{attribute 'GeneratedUsingTerminal: DL-EC1A-0000'}
{attribute addProperty BoxType "DL-EC1A-0000"}
{attribute addProperty Id "ReservedAT %I*DINT4"}
{attribute addProperty CRC "2013026300"}
{attribute addProperty Size "4"}
TYPE
    ID01_Current_Value EXTENDS InputBase_8311D824 :
    STRUCT
        {attribute addProperty Name "Reserved"}
        Reserved AT %I* : DINT;
    END_STRUCT
END_TYPE

(* stored: Version 1.1.0.1, ProductVersion 3.1.4024.12
   DUT ID01_Current_Value: Id {e6f57c76-9e26-0438-224e-f62b823b1ff5} *)
